PROGRAM Comp02_Devices
VAR
END_VAR

END_PROGRAM

(* stored: Version 1.1.0.1, ProductVersion 3.1.4022.11
   POU Comp02_Devices: Id {f02718e1-a717-4016-8298-7cd18f634cd0}, SpecialFunc None *)
